FUNCTION IsItAWorkDay : BOOL

VAR_INPUT
	Day : INT; //Current Day
END_VAR


Day := GVL.DayCounter;
//Checks if the day of the week is a workday
IF Day >= 1 AND Day <= 5 THEN
    IsItAWorkday := TRUE; //Workday (Monday till friday)
ELSE
    IsItAWorkday := FALSE; // Weekend (Saturday and sunday)
END_IF

END_FUNCTION

(* stored: Version 1.1.0.1, ProductVersion 3.1.4024.12
   POU IsItAWorkDay: Id {75519698-d21d-4d12-a3d5-65e39bde2dc3}, SpecialFunc None *)
